(* CoDeSys 2.3.9.9 project: factory_b.pro *)
(* Libraries: standard.lib 4.10.05 11:14:46, Iecsfc.lib 13.4.06 15:51:28, Util.lib 1.6.07 09:40:58, SysLibTime.lib 18.7.05 08:39:56, SysTaskInfo.lib 18.7.05 08:39:56, SysLibMem.lib 18.7.05 08:39:56, SYSLIBCALLBACK.LIB 18.7.05 08:39:56, BusDiag.LIB 27.8.04 14:06:12, SysExt_AC500_V10.lib 1.7.05 15:17:10, SysInt_AC500_V10.LIB 2.6.06 09:49:48, Ethernet_AC500_V10.LIB 28.7.05 11:19:48 *)

(* PLC configuration (modules and I/O channels)
CPU parameters [AC500_CPU] node 0, in %IB0 out %QB0 {AutoRunType = On; ErrLEDType = On; CheckBatteryType = On; OutputsInStopType = Off in hardware and online; StopErrorClassType = No effect; WarmstartOnFK2Type = Off; FloatingPointExceptionType = E2 failure; IOSimulationModeType = Off; NumberRetainSegmentsType = 8; StartRetainM0Type = 0; EndRetainM0Type = 0; StartRetainM1Type = 0; EndRetainM1Type = 0; StartRetainM2Type = 0; EndRetainM2Type = 0; StartRetainM3Type = 0; EndRetainM3Type = 0; StartRetainM4Type = 0; EndRetainM4Type = 0; StartRetainM5Type = 0; EndRetainM5Type = 0; StartRetainM6Type = 0; EndRetainM6Type = 0; StartRetainM7Type = 0; EndRetainM7Type = 0}
AT %IW0 [WordInputNoSpace] Input 0-15
AT %IB0 [ByteInputNoSpace] Input 0-7
S0 AT %IX0.0 [BoolInput] Input 0
S1 AT %IX0.1 [BoolInput] Input 1
S2 AT %IX0.2 [BoolInput] Input 2
S3 AT %IX0.3 [BoolInput] Input 3
S4 AT %IX0.4 [BoolInput] Input 4
S5 AT %IX0.5 [BoolInput] Input 5
S6 AT %IX0.6 [BoolInput] Input 6
S7 AT %IX0.7 [BoolInput] Input 7
AT %IB1 [ByteInputNoSpace] Input 8-15
S8 AT %IX1.0 [BoolInput] Input 8
S9 AT %IX1.1 [BoolInput] Input 9
S10 AT %IX1.2 [BoolInput] Input 10
S11 AT %IX1.3 [BoolInput] Input 11
S12 AT %IX1.4 [BoolInput] Input 12
S13 AT %IX1.5 [BoolInput] Input 13
S14 AT %IX1.6 [BoolInput] Input 14
S15 AT %IX1.7 [BoolInput] Input 15
Digital In/Outputs - Inputs 16-31 [Module_16BitInput_16_31] node 1, in %IB2 out %QB0
  AT %IW1 [WordInputNoSpace] Input 16-31
  AT %IB2 [ByteInputNoSpace] Input 16-23
  AT %IX2.0 [BoolInput] Input 16
  AT %IX2.1 [BoolInput] Input 17
  AT %IX2.2 [BoolInput] Input 18
  AT %IX2.3 [BoolInput] Input 19
  AT %IX2.4 [BoolInput] Input 20
  AT %IX2.5 [BoolInput] Input 21
  AT %IX2.6 [BoolInput] Input 22
  AT %IX2.7 [BoolInput] Input 23
  AT %IB3 [ByteInputNoSpace] Input 24-31
  AT %IX3.0 [BoolInput] Input 24
  AT %IX3.1 [BoolInput] Input 25
  AT %IX3.2 [BoolInput] Input 26
  AT %IX3.3 [BoolInput] Input 27
  AT %IX3.4 [BoolInput] Input 28
  AT %IX3.5 [BoolInput] Input 29
  AT %IX3.6 [BoolInput] Input 30
  AT %IX3.7 [BoolInput] Input 31
AT %QW0 [WordOutputNoSpace] Output 16-31
AT %QB0 [ByteOutputNoSpace] Output 16-23
E0 AT %QX0.0 [BoolOutput] Output 16
E1B AT %QX0.1 [BoolOutput] Output 17
E2B AT %QX0.2 [BoolOutput] Output 18
E3B AT %QX0.3 [BoolOutput] Output 19
E4U AT %QX0.4 [BoolOutput] Output 20
E5B AT %QX0.5 [BoolOutput] Output 21
E6B AT %QX0.6 [BoolOutput] Output 22
E7B AT %QX0.7 [BoolOutput] Output 23
AT %QB1 [ByteOutputNoSpace] Output 24-31
AT %QX1.0 [BoolOutput] Output 24
E1F AT %QX1.1 [BoolOutput] Output 25
E2F AT %QX1.2 [BoolOutput] Output 26
E3F AT %QX1.3 [BoolOutput] Output 27
E4D AT %QX1.4 [BoolOutput] Output 28
E5F AT %QX1.5 [BoolOutput] Output 29
E6F AT %QX1.6 [BoolOutput] Output 30
E7F AT %QX1.7 [BoolOutput] Output 31
Fast counter [Module_2FastCounter] node 3, in %IB4 out %QB2
  AT %ID1 [DWordInput] Istwert/Actual value 1
  AT %ID2 [DWordInput] Istwert/Actual value 2
  AT %IB12 [ByteInputNoBits] Statusbyte/State byte 1
  AT %IB13 [ByteInputNoBits] Statusbyte/State byte 2
  AT %QD1 [DWordOutput] Startwert/Start value 1
  AT %QD2 [DWordOutput] Endwert/End value 1
  AT %QD3 [DWordOutput] Startwert/Start value 2
  AT %QD4 [DWordOutput] Endwert/End value 2
  AT %QB20 [ByteOutputNoBits] Steuerbyte/Control byte 1
  AT %QB21 [ByteOutputNoBits] Steuerbyte/Control byte 2
AT %IW7 [WordInputNoSpace] Input 0-15
AT %IB14 [ByteInputNoSpace] Input 0-7
S16 AT %IX14.0 [BoolInput] Input 0
S17 AT %IX14.1 [BoolInput] Input 1
S18 AT %IX14.2 [BoolInput] Input 2
S19 AT %IX14.3 [BoolInput] Input 3
S20 AT %IX14.4 [BoolInput] Input 4
S21 AT %IX14.5 [BoolInput] Input 5
AT %IX14.6 [BoolInput] Input 6
AT %IX14.7 [BoolInput] Input 7
AT %IB15 [ByteInputNoSpace] Input 8-15
AT %IX15.0 [BoolInput] Input 8
AT %IX15.1 [BoolInput] Input 9
AT %IX15.2 [BoolInput] Input 10
AT %IX15.3 [BoolInput] Input 11
AT %IX15.4 [BoolInput] Input 12
AT %IX15.5 [BoolInput] Input 13
AT %IX15.6 [BoolInput] Input 14
SafetyLine_I215 AT %IX15.7 [BoolInput] Input 15
Digital In/Outputs - Inputs 16-31 [Module_16BitInput_16_31] node 1, in %IB16 out %QB22
  AT %IW8 [WordInputNoSpace] Input 16-31
  AT %IB16 [ByteInputNoSpace] Input 16-23
  AT %IX16.0 [BoolInput] Input 16
  AT %IX16.1 [BoolInput] Input 17
  AT %IX16.2 [BoolInput] Input 18
  AT %IX16.3 [BoolInput] Input 19
  AT %IX16.4 [BoolInput] Input 20
  AT %IX16.5 [BoolInput] Input 21
  AT %IX16.6 [BoolInput] Input 22
  AT %IX16.7 [BoolInput] Input 23
  AT %IB17 [ByteInputNoSpace] Input 24-31
  AT %IX17.0 [BoolInput] Input 24
  AT %IX17.1 [BoolInput] Input 25
  AT %IX17.2 [BoolInput] Input 26
  AT %IX17.3 [BoolInput] Input 27
  AT %IX17.4 [BoolInput] Input 28
  AT %IX17.5 [BoolInput] Input 29
  AT %IX17.6 [BoolInput] Input 30
  AT %IX17.7 [BoolInput] Input 31
AT %QW11 [WordOutputNoSpace] Output 16-31
AT %QB22 [ByteOutputNoSpace] Output 16-23
E8B AT %QX22.0 [BoolOutput] Output 16
AT %QX22.1 [BoolOutput] Output 17
AT %QX22.2 [BoolOutput] Output 18
AT %QX22.3 [BoolOutput] Output 19
AT %QX22.4 [BoolOutput] Output 20
AT %QX22.5 [BoolOutput] Output 21
LOBBY_READY AT %QX22.6 [BoolOutput] Output 22
ALARM AT %QX22.7 [BoolOutput] Output 23
AT %QB23 [ByteOutputNoSpace] Output 24-31
E8F AT %QX23.0 [BoolOutput] Output 24
AT %QX23.1 [BoolOutput] Output 25
AT %QX23.2 [BoolOutput] Output 26
AT %QX23.3 [BoolOutput] Output 27
AT %QX23.4 [BoolOutput] Output 28
AT %QX23.5 [BoolOutput] Output 29
AT %QX23.6 [BoolOutput] Output 30
AT %QX23.7 [BoolOutput] Output 31
AT %ID5 [DWordInput] Istwert/Actual value 1
AT %ID6 [DWordInput] Istwert/Actual value 2
AT %IB28 [ByteInputNoBits] Statusbyte/State byte 1
AT %IB29 [ByteInputNoBits] Statusbyte/State byte 2
AT %QD6 [DWordOutput] Startwert/Start value 1
AT %QD7 [DWordOutput] Endwert/End value 1
AT %QD8 [DWordOutput] Startwert/Start value 2
AT %QD9 [DWordOutput] Endwert/End value 2
AT %QB40 [ByteOutputNoBits] Steuerbyte/Control byte 1
AT %QB41 [ByteOutputNoBits] Steuerbyte/Control byte 2
COM1 - Online access [AC500_COM1_Programming] node 0, in %IB1000 out %QB1000 {COMEnableLoginType = Disabled; COMRTSctrlType = none; COMTLSType = 0; COMCDLYType = 0; COMCharTimeoutType = 0; COMTelEndSelType = none; COMTelEndValCharType = 16#00; COMTelEndValWertType = 0; COMChecksumType = none; COMHandshakeType = none; COMBaudType = 19200; COMParityType = none; COMDataBitType = 8; COMStopBitType = 1}
COM2 - Online access [AC500_COM2_Programming] node 1, in %IB2000 out %QB2000 {COMEnableLoginType = Disabled; COMRTSctrlType = none; COMTLSType = 0; COMCDLYType = 0; COMCharTimeoutType = 0; COMTelEndSelType = none; COMTelEndValCharType = 16#00; COMTelEndValWertType = 0; COMChecksumType = none; COMHandshakeType = none; COMBaudType = 19200; COMParityType = none; COMDataBitType = 8; COMStopBitType = 1}
FBP - none [AC500_FBP_None] node 2, in %IB3000 out %QB3000
MODBUS on TCP/IP [MODBUS_ETH_TCP] node 0, in %IB4000 out %QB4000 {ModbusCouplerOperatingModeType = Master/Slave; COMAdressType = 0; COMDisableWriteStartSeg0Type = 0; COMDisableWriteEndSeg0Type = 0; COMDisableReadStartSeg0Type = 0; COMDisableReadEndSeg0Type = 0; COMDisableWriteStartSeg1Type = 0; COMDisableWriteEndSeg1Type = 0; COMDisableReadStartSeg1Type = 0; COMDisableReadEndSeg1Type = 0}
External - none [AC500_Ext_Empty] node 1, in %IB4000 out %QB4000 {RunConfigFaultType = Yes; MaxWaitRunType = 3000; MinUpdateTimeType = 10; ReserveWord0Type = 0; ReserveWord1Type = 0; ReserveWord2Type = 0}
External - none [AC500_Ext_Empty] node 2, in %IB4000 out %QB4000 {RunConfigFaultType = Yes; MaxWaitRunType = 3000; MinUpdateTimeType = 10; ReserveWord0Type = 0; ReserveWord1Type = 0; ReserveWord2Type = 0}
*)

(* Global variable list: Global_Variables *)
VAR_GLOBAL
	(* Tachometer *)
	TACHO: BOOL := FALSE;
	TACHOTIME: TIME := T#230ms;
	NOT_TACHO:BOOL := FALSE;

	(*Alarms*)
	ROOF_ALARM:BOOL := FALSE;
	STORAGE1_ALARM:BOOL :=FALSE;
	STORAGE2_ALARM:BOOL :=FALSE;

	(*System variables*)
	AutomaticMode:BOOL :=TRUE;
	Emergency:BOOL :=FALSE;
	EffectorFailureTime: TIME := T#500ms;
	SFCInit: BOOL := FALSE;
	SFCReset: BOOL := FALSE;

	(*Variables for the automatic program*)
	START:BOOL :=FALSE;
	STOP:BOOL :=FALSE;
	RUN:BOOL :=FALSE;
	(* LOBBY_READY is a physical communication signal (COM) to factory A *)
	ROOF_READY:BOOL :=FALSE;
	PRESS_READY:BOOL :=FALSE;
	STORAGE1_READY:BOOL :=FALSE;
	STORAGE2_READY:BOOL :=FALSE;
	LOOK_FOR_ROOFS:BOOL :=FALSE;
	NO_ROOFS:BOOL :=FALSE;
	START_PRESS_UP:BOOL :=FALSE;
	START_PRESS_DOWN:BOOL :=FALSE;
	STOP_PRESS:BOOL :=FALSE;
	(* Faulty car flag *)
	FAULTY_CAR:BOOL := FALSE;
	GOOD_CAR:BOOL := FALSE;
	(* Assembly line variables *)
	E0A:BOOL := FALSE;
	E0B:BOOL := FALSE;
	E0C:BOOL := FALSE;
	E0D:BOOL := FALSE;
	E0E:BOOL := FALSE;
	E0F:BOOL := FALSE;
	(* Safe motor variables*)
	E0AS:BOOL :=FALSE;
	E1FS:BOOL := FALSE;
	E1BS:BOOL := FALSE;
	E2FS:BOOL := FALSE;
	E2BS:BOOL := FALSE;
	E3FS:BOOL := FALSE;
	E3BS:BOOL := FALSE;
	E4US:BOOL := FALSE;
	E4DS:BOOL := FALSE;
	E5FS:BOOL := FALSE;
	E5BS:BOOL := FALSE;
	E6FS:BOOL := FALSE;
	E6BS:BOOL := FALSE;
	E7FS:BOOL := FALSE;
	E7BS:BOOL := FALSE;
	E8FS:BOOL := FALSE;
	E8BS:BOOL := FALSE;
	(* Car detection variables *)
	LOOK_FOR_CAR_LOBBY:BOOL :=FALSE;
	CAR_ARRIVED_LOBBY:BOOL :=FALSE;
	LOOK_FOR_CAR_ROOF:BOOL :=FALSE;
	CAR_ARRIVED_ROOF:BOOL :=FALSE;
	LOOK_FOR_CAR_PRESS:BOOL :=FALSE;
	CAR_ARRIVED_PRESS:BOOL :=FALSE;
	LOOK_FOR_CAR_STORAGE1:BOOL :=FALSE;
	CAR_DETECTED_STORAGE1:BOOL :=FALSE;
	CAR_ARRIVED_STORAGE1:BOOL :=FALSE;
	LOOK_FOR_CAR_STORAGE2:BOOL :=FALSE;
	CAR_DETECTED_STORAGE2:BOOL :=FALSE;
	CAR_ARRIVED_STORAGE2:BOOL :=FALSE;
END_VAR

(* POU PLC_PRG, LD *)
PROGRAM PLC_PRG
VAR
	automaticFalling: F_TRIG;
	automaticRising: R_TRIG;
	TachoTimer1: TON;
	TachoTimer2: TON;
	EffectorFailure: BOOL;
	E1FailureTimer1: TON;
	E1FailureTimer2: TON;
	E1Failure: BOOL;
	E2FailureTimer1: TON;
	E2FailureTimer2: TON;
	E2Failure: BOOL;
	E3FailureTimer1: TON;
	E3FailureTimer2: TON;
	E3Failure: BOOL;
	E4FailureTimer1: TON;
	E4FailureTimer2: TON;
	E4Failure: BOOL;
	E5FailureTimer1: TON;
	E5FailureTimer2: TON;
	E5Failure: BOOL;
	E6FailureTimer1: TON;
	E6FailureTimer2: TON;
	E6Failure: BOOL;
	E7FailureTimer1: TON;
	E7FailureTimer2: TON;
	E7Failure: BOOL;
	E8FailureTimer1: TON;
	E8FailureTimer2: TON;
	E8Failure: BOOL;
END_VAR
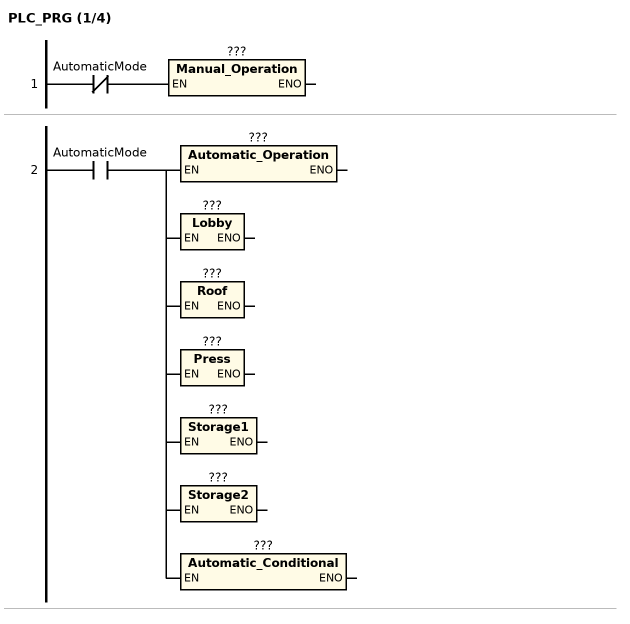
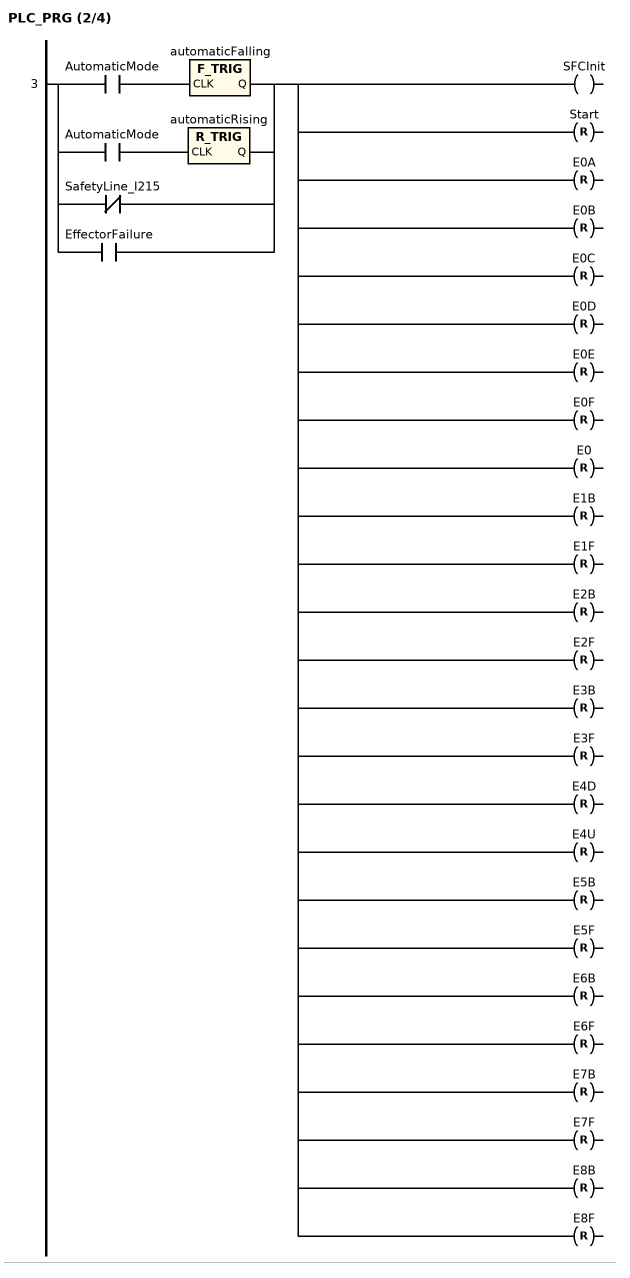
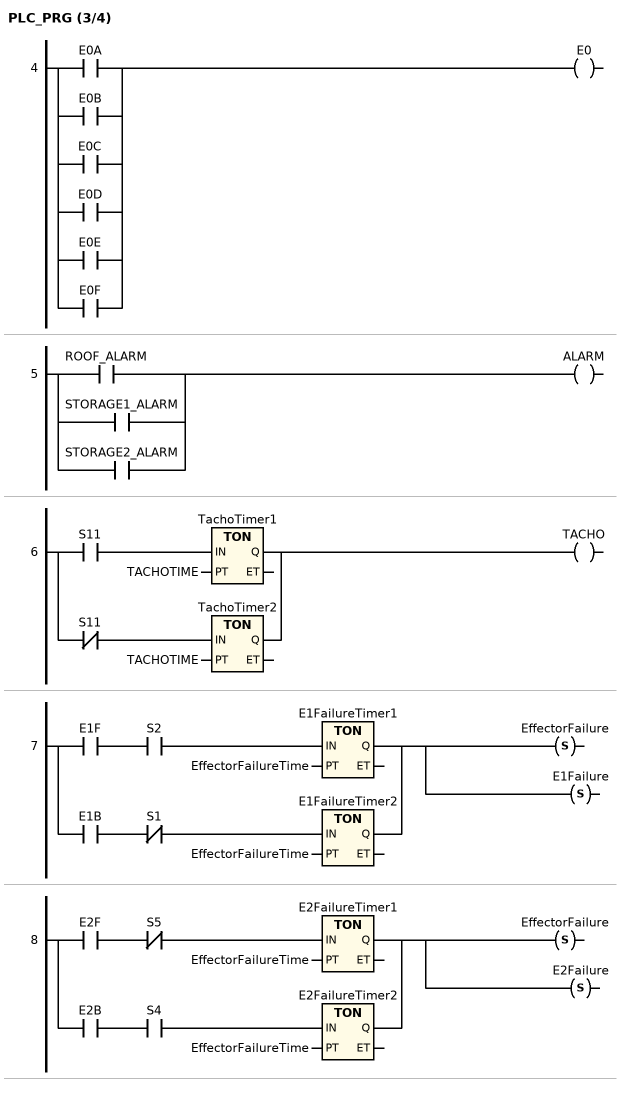
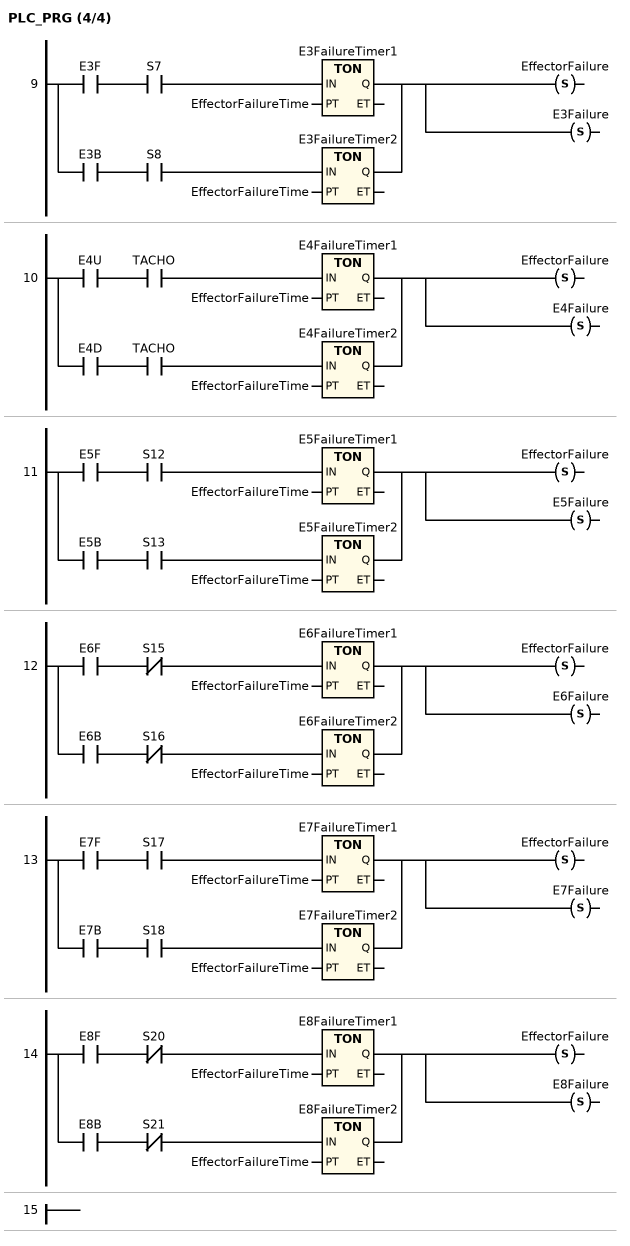
_LD_ (* Ladder Diagram *)
NETWORK 1
	[/AutomaticMode]
		EN --- ???:Manual_Operation()
NETWORK 2
	[AutomaticMode]
		EN --- ???:Automatic_Operation()
		EN --- ???:Lobby()
		EN --- ???:Roof()
		EN --- ???:Press()
		EN --- ???:Storage1()
		EN --- ???:Storage2()
		EN --- ???:Automatic_Conditional()
NETWORK 3
	{ [AutomaticMode] - automaticFalling:F_TRIG(CLK: *) | [AutomaticMode] - automaticRising:R_TRIG(CLK: *) | [/SafetyLine_I215] | [EffectorFailure] } --- (SFCInit) (R Start) (R E0A) (R E0B) (R E0C) (R E0D) (R E0E) (R E0F) (R E0) (R E1B) (R E1F) (R E2B) (R E2F) (R E3B) (R E3F) (R E4D) (R E4U) (R E5B) (R E5F) (R E6B) (R E6F) (R E7B) (R E7F) (R E8B) (R E8F)
NETWORK 4
	{ [E0A] | [E0B] | [E0C] | [E0D] | [E0E] | [E0F] } --- (E0)
NETWORK 5
	{ [ROOF_ALARM] | [STORAGE1_ALARM] | [STORAGE2_ALARM] } --- (ALARM)
NETWORK 6
	{ [S11] - TachoTimer1:TON(IN: *, PT: TACHOTIME) | [/S11] - TachoTimer2:TON(IN: *, PT: TACHOTIME) } --- (TACHO)
NETWORK 7
	{ [E1F] - [S2] - E1FailureTimer1:TON(IN: *, PT: EffectorFailureTime) | [E1B] - [/S1] - E1FailureTimer2:TON(IN: *, PT: EffectorFailureTime) } --- (S EffectorFailure) (S E1Failure)
NETWORK 8
	{ [E2F] - [/S5] - E2FailureTimer1:TON(IN: *, PT: EffectorFailureTime) | [E2B] - [S4] - E2FailureTimer2:TON(IN: *, PT: EffectorFailureTime) } --- (S EffectorFailure) (S E2Failure)
NETWORK 9
	{ [E3F] - [S7] - E3FailureTimer1:TON(IN: *, PT: EffectorFailureTime) | [E3B] - [S8] - E3FailureTimer2:TON(IN: *, PT: EffectorFailureTime) } --- (S EffectorFailure) (S E3Failure)
NETWORK 10
	{ [E4U] - [TACHO] - E4FailureTimer1:TON(IN: *, PT: EffectorFailureTime) | [E4D] - [TACHO] - E4FailureTimer2:TON(IN: *, PT: EffectorFailureTime) } --- (S EffectorFailure) (S E4Failure)
NETWORK 11
	{ [E5F] - [S12] - E5FailureTimer1:TON(IN: *, PT: EffectorFailureTime) | [E5B] - [S13] - E5FailureTimer2:TON(IN: *, PT: EffectorFailureTime) } --- (S EffectorFailure) (S E5Failure)
NETWORK 12
	{ [E6F] - [/S15] - E6FailureTimer1:TON(IN: *, PT: EffectorFailureTime) | [E6B] - [/S16] - E6FailureTimer2:TON(IN: *, PT: EffectorFailureTime) } --- (S EffectorFailure) (S E6Failure)
NETWORK 13
	{ [E7F] - [S17] - E7FailureTimer1:TON(IN: *, PT: EffectorFailureTime) | [E7B] - [S18] - E7FailureTimer2:TON(IN: *, PT: EffectorFailureTime) } --- (S EffectorFailure) (S E7Failure)
NETWORK 14
	{ [E8F] - [/S20] - E8FailureTimer1:TON(IN: *, PT: EffectorFailureTime) | [E8B] - [/S21] - E8FailureTimer2:TON(IN: *, PT: EffectorFailureTime) } --- (S EffectorFailure) (S E8Failure)
NETWORK 15
	*
_END_LD_
(* the same logic as Structured Text *)
(* Network 1: see the listing above *)
(* Network 2: see the listing above *)
(* Network 3 *)
automaticFalling(CLK := AutomaticMode);
automaticRising(CLK := AutomaticMode);
SFCInit := automaticFalling.Q OR automaticRising.Q OR NOT SafetyLine_I215 OR EffectorFailure;
IF SFCInit THEN Start := FALSE; E0A := FALSE; E0B := FALSE; E0C := FALSE; E0D := FALSE; E0E := FALSE; E0F := FALSE; E0 := FALSE; E1B := FALSE; E1F := FALSE; E2B := FALSE; E2F := FALSE; E3B := FALSE; E3F := FALSE; E4D := FALSE; E4U := FALSE; E5B := FALSE; E5F := FALSE; E6B := FALSE; E6F := FALSE; E7B := FALSE; E7F := FALSE; E8B := FALSE; E8F := FALSE; END_IF;
(* Network 4 *)
E0 := E0A OR E0B OR E0C OR E0D OR E0E OR E0F;
(* Network 5 *)
ALARM := ROOF_ALARM OR STORAGE1_ALARM OR STORAGE2_ALARM;
(* Network 6 *)
TachoTimer1(IN := S11, PT := TACHOTIME);
TachoTimer2(IN := NOT S11, PT := TACHOTIME);
TACHO := TachoTimer1.Q OR TachoTimer2.Q;
(* Network 7 *)
E1FailureTimer1(IN := E1F AND S2, PT := EffectorFailureTime);
E1FailureTimer2(IN := E1B AND NOT S1, PT := EffectorFailureTime);
IF E1FailureTimer1.Q OR E1FailureTimer2.Q THEN EffectorFailure := TRUE; E1Failure := TRUE; END_IF;
(* Network 8 *)
E2FailureTimer1(IN := E2F AND NOT S5, PT := EffectorFailureTime);
E2FailureTimer2(IN := E2B AND S4, PT := EffectorFailureTime);
IF E2FailureTimer1.Q OR E2FailureTimer2.Q THEN EffectorFailure := TRUE; E2Failure := TRUE; END_IF;
(* Network 9 *)
E3FailureTimer1(IN := E3F AND S7, PT := EffectorFailureTime);
E3FailureTimer2(IN := E3B AND S8, PT := EffectorFailureTime);
IF E3FailureTimer1.Q OR E3FailureTimer2.Q THEN EffectorFailure := TRUE; E3Failure := TRUE; END_IF;
(* Network 10 *)
E4FailureTimer1(IN := E4U AND TACHO, PT := EffectorFailureTime);
E4FailureTimer2(IN := E4D AND TACHO, PT := EffectorFailureTime);
IF E4FailureTimer1.Q OR E4FailureTimer2.Q THEN EffectorFailure := TRUE; E4Failure := TRUE; END_IF;
(* Network 11 *)
E5FailureTimer1(IN := E5F AND S12, PT := EffectorFailureTime);
E5FailureTimer2(IN := E5B AND S13, PT := EffectorFailureTime);
IF E5FailureTimer1.Q OR E5FailureTimer2.Q THEN EffectorFailure := TRUE; E5Failure := TRUE; END_IF;
(* Network 12 *)
E6FailureTimer1(IN := E6F AND NOT S15, PT := EffectorFailureTime);
E6FailureTimer2(IN := E6B AND NOT S16, PT := EffectorFailureTime);
IF E6FailureTimer1.Q OR E6FailureTimer2.Q THEN EffectorFailure := TRUE; E6Failure := TRUE; END_IF;
(* Network 13 *)
E7FailureTimer1(IN := E7F AND S17, PT := EffectorFailureTime);
E7FailureTimer2(IN := E7B AND S18, PT := EffectorFailureTime);
IF E7FailureTimer1.Q OR E7FailureTimer2.Q THEN EffectorFailure := TRUE; E7Failure := TRUE; END_IF;
(* Network 14 *)
E8FailureTimer1(IN := E8F AND NOT S20, PT := EffectorFailureTime);
E8FailureTimer2(IN := E8B AND NOT S21, PT := EffectorFailureTime);
IF E8FailureTimer1.Q OR E8FailureTimer2.Q THEN EffectorFailure := TRUE; E8Failure := TRUE; END_IF;
(* Network 15: see the listing above *)
END_PROGRAM

(* POU Manual_Operation, SFC *)
(*FactoryB*)

PROGRAM Manual_Operation
VAR
	StorageAlarmTime:TIME :=T#2S;
	(*E0: Assembly line*)
	(*Not in SFC.Using  E0AssemblyLine_O16 directly*)
	(*E1: LobbyBar*)
	buttonE1Fwd:BOOL :=FALSE;
	buttonE1Bwd:BOOL :=FALSE;
	(*E2: RoofPusher*)
	buttonE2Fwd:BOOL :=FALSE;
	buttonE2Bwd:BOOL :=FALSE;
	(*E3: RoofBar*)
	buttonE3Fwd:BOOL :=FALSE;
	buttonE3Bwd:BOOL :=FALSE;
	(*E4: Press*)
	buttonE4Press:BOOL :=FALSE;
	PressStarted: BOOL := FALSE;
	(*E5: Press bar*)
	buttonE5Fwd:BOOL :=FALSE;
	buttonE5Bwd:BOOL :=FALSE;
	(*E6: Storage1Pusher*)
	buttonE6Fwd:BOOL :=FALSE;
	buttonE6Bwd:BOOL :=FALSE;
	TimeOutStorage1: BOOL;
	(*E7: Storage1Bar*)
	buttonE7Fwd:BOOL :=FALSE;
	buttonE7Bwd:BOOL :=FALSE;
	(*E8: Storage2Pusher*)
	buttonE8Fwd:BOOL :=FALSE;
	buttonE8Bwd:BOOL :=FALSE;
	TimeOutStorage2: BOOL;
END_VAR
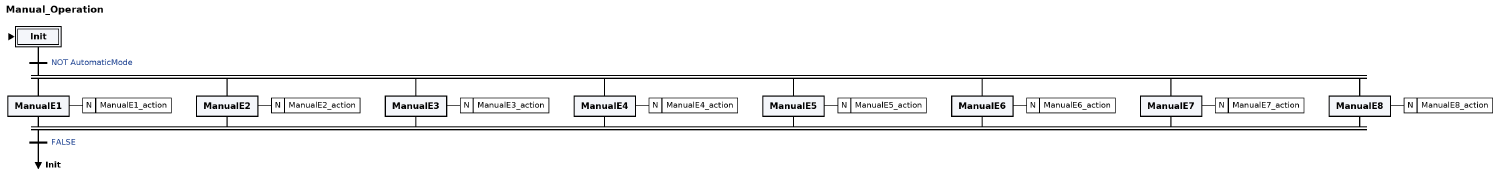
INITIAL_STEP Init:
END_STEP
TRANSITION FROM Init TO (ManualE1, ManualE2, ManualE3, ManualE4, ManualE5, ManualE6, ManualE7, ManualE8) := NOT AutomaticMode;
END_TRANSITION
STEP ManualE1:
	ManualE1_action(N);
END_STEP
STEP ManualE2:
	ManualE2_action(N);
END_STEP
STEP ManualE3:
	ManualE3_action(N);
END_STEP
STEP ManualE4:
	ManualE4_action(N);
END_STEP
STEP ManualE5:
	ManualE5_action(N);
END_STEP
STEP ManualE6:
	ManualE6_action(N);
END_STEP
STEP ManualE7:
	ManualE7_action(N);
END_STEP
STEP ManualE8:
	ManualE8_action(N);
END_STEP
TRANSITION FROM (ManualE1, ManualE2, ManualE3, ManualE4, ManualE5, ManualE6, ManualE7, ManualE8) TO Init := FALSE;
END_TRANSITION

ACTION ManualE1_action:
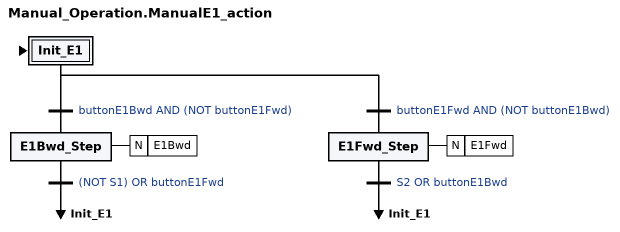
INITIAL_STEP Init_E1:
END_STEP
TRANSITION FROM Init_E1 TO E1Bwd_Step := buttonE1Bwd AND (NOT buttonE1Fwd);
END_TRANSITION
TRANSITION FROM Init_E1 TO E1Fwd_Step := buttonE1Fwd AND (NOT buttonE1Bwd);
END_TRANSITION
STEP E1Bwd_Step:
	E1Bwd(N);
END_STEP
TRANSITION FROM E1Bwd_Step TO Init_E1 := (NOT S1) OR buttonE1Fwd;
END_TRANSITION
STEP E1Fwd_Step:
	E1Fwd(N);
END_STEP
TRANSITION FROM E1Fwd_Step TO Init_E1 := S2 OR buttonE1Bwd;
END_TRANSITION
END_ACTION

ACTION ManualE2_action:
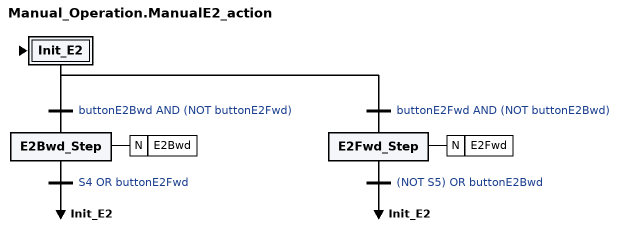
INITIAL_STEP Init_E2:
END_STEP
TRANSITION FROM Init_E2 TO E2Bwd_Step := buttonE2Bwd AND (NOT buttonE2Fwd);
END_TRANSITION
TRANSITION FROM Init_E2 TO E2Fwd_Step := buttonE2Fwd AND (NOT buttonE2Bwd);
END_TRANSITION
STEP E2Bwd_Step:
	E2Bwd(N);
END_STEP
TRANSITION FROM E2Bwd_Step TO Init_E2 := S4 OR buttonE2Fwd;
END_TRANSITION
STEP E2Fwd_Step:
	E2Fwd(N);
END_STEP
TRANSITION FROM E2Fwd_Step TO Init_E2 := (NOT S5) OR buttonE2Bwd;
END_TRANSITION
END_ACTION

ACTION ManualE3_action:
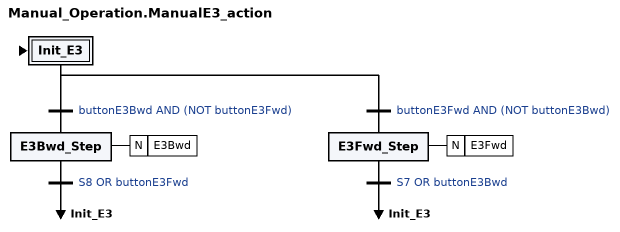
INITIAL_STEP Init_E3:
END_STEP
TRANSITION FROM Init_E3 TO E3Bwd_Step := buttonE3Bwd AND (NOT buttonE3Fwd);
END_TRANSITION
TRANSITION FROM Init_E3 TO E3Fwd_Step := buttonE3Fwd AND (NOT buttonE3Bwd);
END_TRANSITION
STEP E3Bwd_Step:
	E3Bwd(N);
END_STEP
TRANSITION FROM E3Bwd_Step TO Init_E3 := S8 OR buttonE3Fwd;
END_TRANSITION
STEP E3Fwd_Step:
	E3Fwd(N);
END_STEP
TRANSITION FROM E3Fwd_Step TO Init_E3 := S7 OR buttonE3Bwd;
END_TRANSITION
END_ACTION

ACTION ManualE4_action:
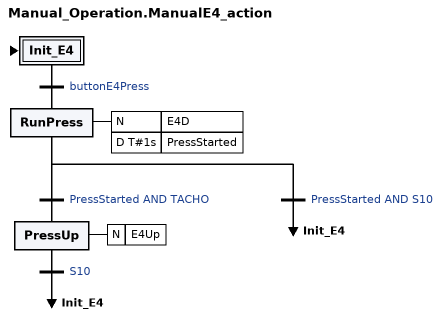
INITIAL_STEP Init_E4:
END_STEP
TRANSITION FROM Init_E4 TO RunPress := buttonE4Press;
END_TRANSITION
STEP RunPress:
	E4D(N);
	PressStarted(D, T#1s);
END_STEP
TRANSITION FROM RunPress TO PressUp := PressStarted AND TACHO;
END_TRANSITION
TRANSITION FROM RunPress TO Init_E4 := PressStarted AND S10;
END_TRANSITION
STEP PressUp:
	E4Up(N);
END_STEP
TRANSITION FROM PressUp TO Init_E4 := S10;
END_TRANSITION
END_ACTION

ACTION ManualE5_action:
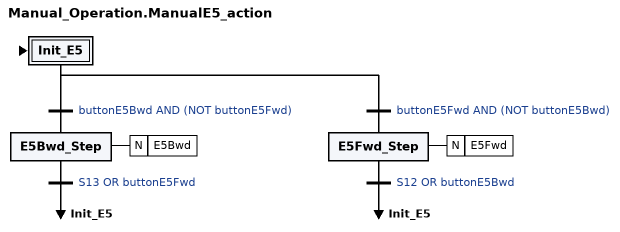
INITIAL_STEP Init_E5:
END_STEP
TRANSITION FROM Init_E5 TO E5Bwd_Step := buttonE5Bwd AND (NOT buttonE5Fwd);
END_TRANSITION
TRANSITION FROM Init_E5 TO E5Fwd_Step := buttonE5Fwd AND (NOT buttonE5Bwd);
END_TRANSITION
STEP E5Bwd_Step:
	E5Bwd(N);
END_STEP
TRANSITION FROM E5Bwd_Step TO Init_E5 := S13 OR buttonE5Fwd;
END_TRANSITION
STEP E5Fwd_Step:
	E5Fwd(N);
END_STEP
TRANSITION FROM E5Fwd_Step TO Init_E5 := S12 OR buttonE5Bwd;
END_TRANSITION
END_ACTION

ACTION ManualE6_action:
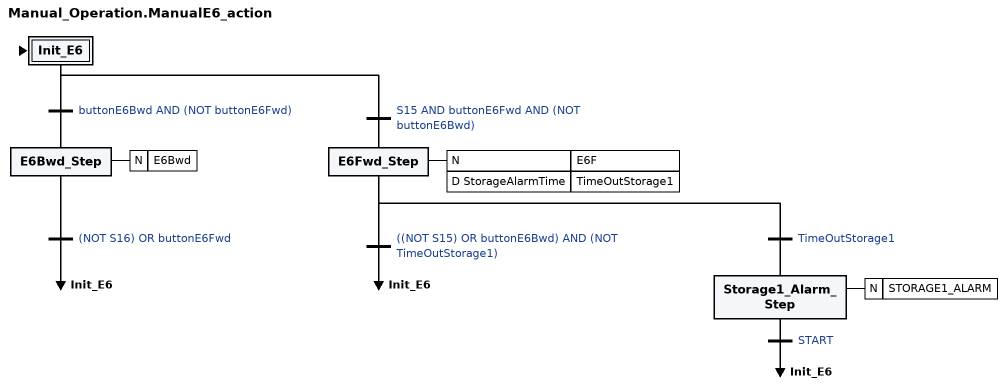
INITIAL_STEP Init_E6:
END_STEP
TRANSITION FROM Init_E6 TO E6Bwd_Step := buttonE6Bwd AND (NOT buttonE6Fwd);
END_TRANSITION
TRANSITION FROM Init_E6 TO E6Fwd_Step := S15 AND buttonE6Fwd AND (NOT buttonE6Bwd);
END_TRANSITION
STEP E6Bwd_Step:
	E6Bwd(N);
END_STEP
TRANSITION FROM E6Bwd_Step TO Init_E6 := (NOT S16) OR buttonE6Fwd;
END_TRANSITION
STEP E6Fwd_Step:
	E6F(N);
	TimeOutStorage1(D, StorageAlarmTime);
END_STEP
TRANSITION FROM E6Fwd_Step TO Init_E6 := ((NOT S15) OR buttonE6Bwd) AND (NOT TimeOutStorage1);
END_TRANSITION
TRANSITION FROM E6Fwd_Step TO Storage1_Alarm_Step := TimeOutStorage1;
END_TRANSITION
STEP Storage1_Alarm_Step:
	STORAGE1_ALARM(N);
END_STEP
TRANSITION FROM Storage1_Alarm_Step TO Init_E6 := START;
END_TRANSITION
END_ACTION

ACTION ManualE7_action:
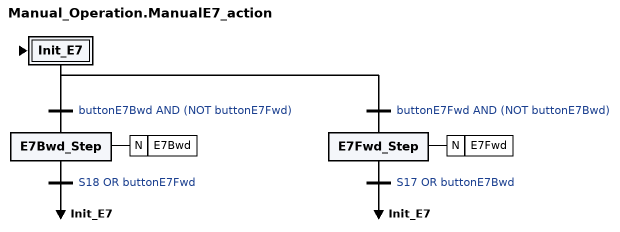
INITIAL_STEP Init_E7:
END_STEP
TRANSITION FROM Init_E7 TO E7Bwd_Step := buttonE7Bwd AND (NOT buttonE7Fwd);
END_TRANSITION
TRANSITION FROM Init_E7 TO E7Fwd_Step := buttonE7Fwd AND (NOT buttonE7Bwd);
END_TRANSITION
STEP E7Bwd_Step:
	E7Bwd(N);
END_STEP
TRANSITION FROM E7Bwd_Step TO Init_E7 := S18 OR buttonE7Fwd;
END_TRANSITION
STEP E7Fwd_Step:
	E7Fwd(N);
END_STEP
TRANSITION FROM E7Fwd_Step TO Init_E7 := S17 OR buttonE7Bwd;
END_TRANSITION
END_ACTION

ACTION ManualE8_action:
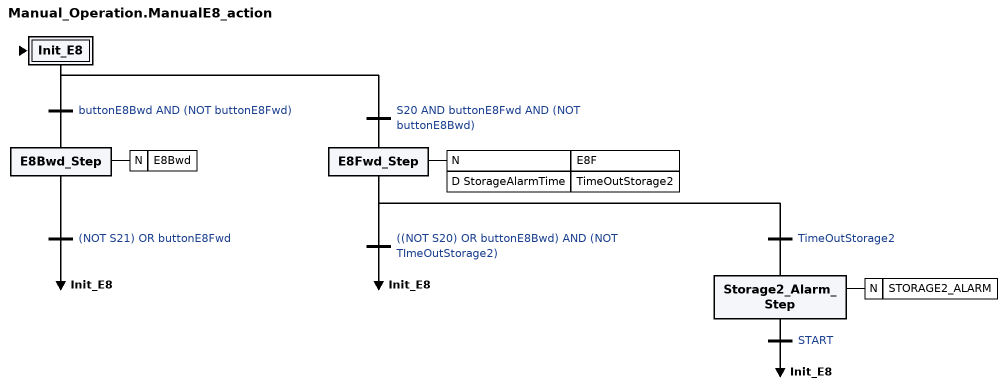
INITIAL_STEP Init_E8:
END_STEP
TRANSITION FROM Init_E8 TO E8Bwd_Step := buttonE8Bwd AND (NOT buttonE8Fwd);
END_TRANSITION
TRANSITION FROM Init_E8 TO E8Fwd_Step := S20 AND buttonE8Fwd AND (NOT buttonE8Bwd);
END_TRANSITION
STEP E8Bwd_Step:
	E8Bwd(N);
END_STEP
TRANSITION FROM E8Bwd_Step TO Init_E8 := (NOT S21) OR buttonE8Fwd;
END_TRANSITION
STEP E8Fwd_Step:
	E8F(N);
	TimeOutStorage2(D, StorageAlarmTime);
END_STEP
TRANSITION FROM E8Fwd_Step TO Init_E8 := ((NOT S20) OR buttonE8Bwd) AND (NOT TImeOutStorage2);
END_TRANSITION
TRANSITION FROM E8Fwd_Step TO Storage2_Alarm_Step := TimeOutStorage2;
END_TRANSITION
STEP Storage2_Alarm_Step:
	STORAGE2_ALARM(N);
END_STEP
TRANSITION FROM Storage2_Alarm_Step TO Init_E8 := START;
END_TRANSITION
END_ACTION
END_PROGRAM
ACTION E1Bwd:
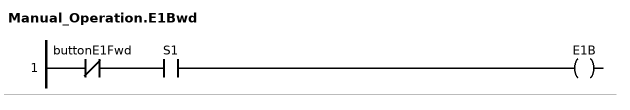
_LD_ (* Ladder Diagram *)
NETWORK 1
	[/buttonE1Fwd] - [S1] --- (E1B)
_END_LD_
(* the same logic as Structured Text *)
(* Network 1 *)
E1B := NOT buttonE1Fwd AND S1;
END_ACTION
ACTION E1Fwd:
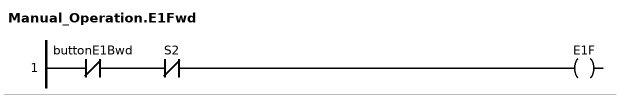
_LD_ (* Ladder Diagram *)
NETWORK 1
	[/buttonE1Bwd] - [/S2] --- (E1F)
_END_LD_
(* the same logic as Structured Text *)
(* Network 1 *)
E1F := NOT buttonE1Bwd AND NOT S2;
END_ACTION
ACTION E2Bwd:
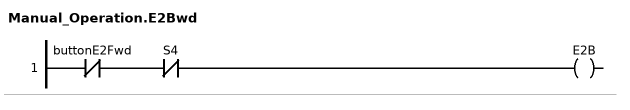
_LD_ (* Ladder Diagram *)
NETWORK 1
	[/buttonE2Fwd] - [/S4] --- (E2B)
_END_LD_
(* the same logic as Structured Text *)
(* Network 1 *)
E2B := NOT buttonE2Fwd AND NOT S4;
END_ACTION
ACTION E2Fwd:
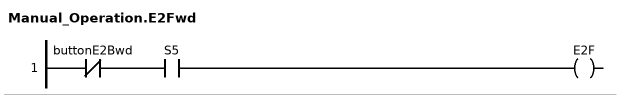
_LD_ (* Ladder Diagram *)
NETWORK 1
	[/buttonE2Bwd] - [S5] --- (E2F)
_END_LD_
(* the same logic as Structured Text *)
(* Network 1 *)
E2F := NOT buttonE2Bwd AND S5;
END_ACTION
ACTION E3Bwd:
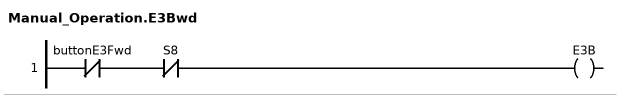
_LD_ (* Ladder Diagram *)
NETWORK 1
	[/buttonE3Fwd] - [/S8] --- (E3B)
_END_LD_
(* the same logic as Structured Text *)
(* Network 1 *)
E3B := NOT buttonE3Fwd AND NOT S8;
END_ACTION
ACTION E3Fwd:
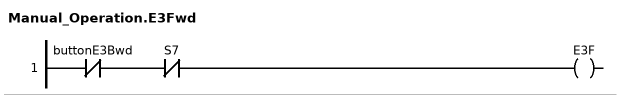
_LD_ (* Ladder Diagram *)
NETWORK 1
	[/buttonE3Bwd] - [/S7] --- (E3F)
_END_LD_
(* the same logic as Structured Text *)
(* Network 1 *)
E3F := NOT buttonE3Bwd AND NOT S7;
END_ACTION
ACTION E4Up:
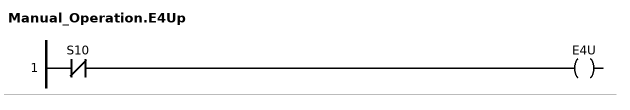
_LD_ (* Ladder Diagram *)
NETWORK 1
	[/S10] --- (E4U)
_END_LD_
(* the same logic as Structured Text *)
(* Network 1 *)
E4U := NOT S10;
END_ACTION
ACTION E5Bwd:
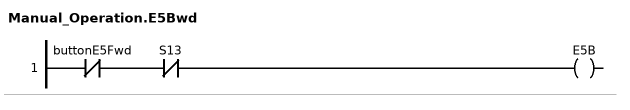
_LD_ (* Ladder Diagram *)
NETWORK 1
	[/buttonE5Fwd] - [/S13] --- (E5B)
_END_LD_
(* the same logic as Structured Text *)
(* Network 1 *)
E5B := NOT buttonE5Fwd AND NOT S13;
END_ACTION
ACTION E5Fwd:
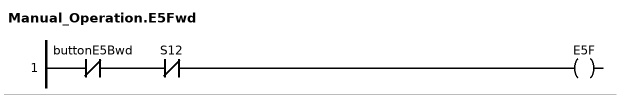
_LD_ (* Ladder Diagram *)
NETWORK 1
	[/buttonE5Bwd] - [/S12] --- (E5F)
_END_LD_
(* the same logic as Structured Text *)
(* Network 1 *)
E5F := NOT buttonE5Bwd AND NOT S12;
END_ACTION
ACTION E6Bwd:
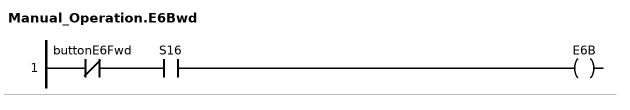
_LD_ (* Ladder Diagram *)
NETWORK 1
	[/buttonE6Fwd] - [S16] --- (E6B)
_END_LD_
(* the same logic as Structured Text *)
(* Network 1 *)
E6B := NOT buttonE6Fwd AND S16;
END_ACTION
ACTION E7Bwd:
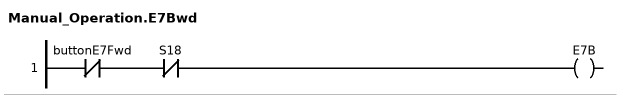
_LD_ (* Ladder Diagram *)
NETWORK 1
	[/buttonE7Fwd] - [/S18] --- (E7B)
_END_LD_
(* the same logic as Structured Text *)
(* Network 1 *)
E7B := NOT buttonE7Fwd AND NOT S18;
END_ACTION
ACTION E7Fwd:
